//tcUNIT_GVL: Global variables used in tcUNIT tests.
{attribute 'qualified_only'}
VAR_GLOBAL CONSTANT
//Constants for axis defaults.
fDEFAULT_VELOCITY: LREAL := 0.0;
fDEFAULT_ACCELERATION: LREAL := 0.0;
fDEFAULT_DECCELERATION: LREAL := 0.0;
fDEFAULT_POSITION: LREAL := 0.0;
fDEFAULT_TARGET_VELOCITY: LREAL := 1.0;
fDEFAULT_TARGET_ACCELERATION: LREAL := 0.5;
fDEFAULT_TARGET_DECCELERATION: LREAL := 0.5;
fDEFAULT_TARGET_POSITION: LREAL := 10.0;
fDEFAULT_TARGET_OVERRIDE: LREAL := 100;
nMAX_MASTERS : UINT := 4;
END_VAR

VAR_GLOBAL
END_VAR

(* stored: Version 1.1.0.1, ProductVersion 3.1.4024.0
   GVL tcUNIT_GVL: Id {4b23d6c9-6a88-40b7-9bf4-d55c4dfd4246} *)
